Staubli VAL3: iTeste.pgx

public program iTeste(num& nNum[] (dimensions=1))
begin
end
